// TIA Portal V20 export
FUNCTION_BLOCK "LER_SimAxis+"   // FB90, LAD
// stored: Access Published, MemoryReserve 100, SetENOAutomatically false
   VAR_INPUT
      axisActualPos { ExternalAccessible := 'False'; ExternalVisible := 'False'; ExternalWritable := 'False'} : LReal;
      pixel { ExternalAccessible := 'False'; ExternalVisible := 'False'; ExternalWritable := 'False'} : Int := 0;
      startposition : LReal;
      endposition : LReal;
      Maxipixel : Int;
      Minpixel : Int;
   END_VAR
   VAR_OUTPUT
      simHmiAxis { ExternalAccessible := 'False'; ExternalVisible := 'False'; ExternalWritable := 'False'} : "LER_typeSimLinearAxis";
   END_VAR
   VAR
      axisActualPosReal : Real;
      t_hmiTravleDistance { ExternalAccessible := 'False'; ExternalVisible := 'False'; ExternalWritable := 'False'} : Int;
   END_VAR
BEGIN

REGION Network 2
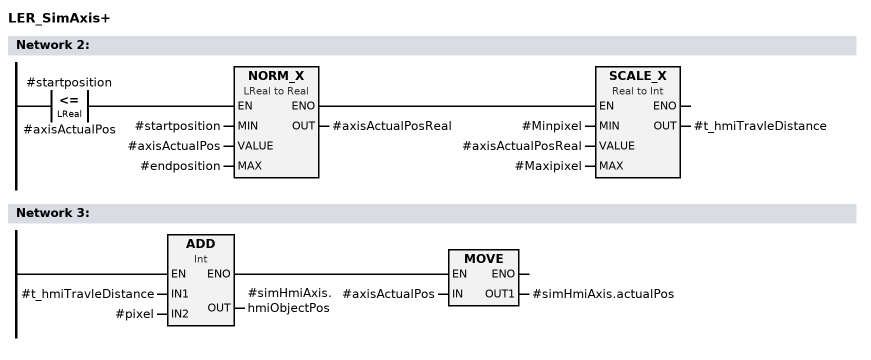
   RUNG wire#powerrail
      { S7_Templates := "SrcType := LReal" } LE_Contact(in1 := #startposition, in2 := #axisActualPos)
      { S7_Templates := "[SrcType := LReal, DestType := Real]" } Normalize(min := #startposition, value := #axisActualPos, max := #endposition, out => #axisActualPosReal)
      { S7_Templates := "[SrcType := Real, DestType := Int]" } Scale(min := #Minpixel, value := #axisActualPosReal, max := #Maxipixel, out => #t_hmiTravleDistance)
   END_RUNG
   // the same network as SCL:
   IF #startposition <= #axisActualPos THEN
       #axisActualPosReal := NORM_X(MIN := #startposition, VALUE := #axisActualPos, MAX := #endposition);
       #t_hmiTravleDistance := SCALE_X(MIN := #Minpixel, VALUE := #axisActualPosReal, MAX := #Maxipixel);
   END_IF;
END_REGION

REGION Network 3
   RUNG wire#powerrail
      { S7_Templates := "SrcType := Int" } Add(in1 := #t_hmiTravleDistance, in2 := #pixel, out => #simHmiAxis.hmiObjectPos)
      Move(in := #axisActualPos, out1 => #simHmiAxis.actualPos)
   END_RUNG
   // the same network as SCL:
   #simHmiAxis.hmiObjectPos := #t_hmiTravleDistance + #pixel;
   #simHmiAxis.actualPos := #axisActualPos;
END_REGION
END_FUNCTION_BLOCK
